FUNCTION_BLOCK FB_SchmittTrigger
VAR_INPUT
    fInput : REAL;
    fLowThreshold : REAL := 0.3;
    fHighThreshold : REAL := 0.7;
END_VAR
VAR_OUTPUT
    bState : BOOL;
END_VAR

METHOD Step : BOOL
;
END_METHOD

END_FUNCTION_BLOCK

(* stored: Version 1.1.0.1
   POU FB_SchmittTrigger: Id {c39c0c34-cb35-47af-b6a2-847e3a2e2173}, SpecialFunc None
   Method Step: Id {a8c636f3-d0be-4cbf-8eba-f6a1227bce65} *)
